FUNCTION_BLOCK ButtonColorChanger (* Composite FB wrapping other FBs *)
  (* Standard: 61499-2 *)
  (* Version 1.0, 2022-08-01, franz *)
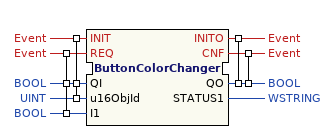
  EVENT_INPUT
    INIT WITH QI, u16ObjId; (* Initialization Request *)
    REQ WITH QI, I1; (* Normal Execution Request *)
  END_EVENT
  EVENT_OUTPUT
    INITO WITH QO; (* Initialization Confirm *)
    CNF WITH QO; (* Execution Confirmation *)
  END_EVENT
  VAR_INPUT
    QI : BOOL; (* Input event qualifier *)
    u16ObjId : UINT; (* Object ID *)
    I1 : BOOL;
  END_VAR
  VAR_OUTPUT
    QO : BOOL; (* Output event qualifier *)
    STATUS1 : WSTRING;
  END_VAR
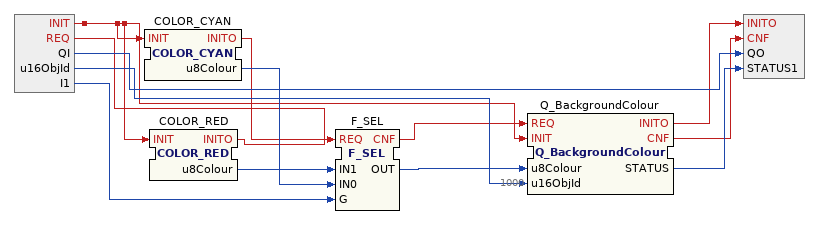
  FBS
    Q_BackgroundColour : Q_BackgroundColour(u16ObjId := 1000);
    F_SEL : F_SEL;
    COLOR_RED : COLOR_RED;
    COLOR_CYAN : COLOR_CYAN;
  END_FBS
  EVENT_CONNECTIONS
    F_SEL.CNF TO Q_BackgroundColour.REQ;
    COLOR_CYAN.INITO TO F_SEL.REQ;
    COLOR_RED.INITO TO F_SEL.REQ;
    Q_BackgroundColour.INITO TO INITO;
    INIT TO COLOR_CYAN.INIT;
    INIT TO COLOR_RED.INIT;
    Q_BackgroundColour.CNF TO CNF;
    REQ TO F_SEL.REQ;
    INIT TO Q_BackgroundColour.INIT;
  END_CONNECTIONS
  DATA_CONNECTIONS
    COLOR_RED.u8Colour TO F_SEL.IN1;
    COLOR_CYAN.u8Colour TO F_SEL.IN0;
    F_SEL.OUT TO Q_BackgroundColour.u8Colour;
    u16ObjId TO Q_BackgroundColour.u16ObjId;
    Q_BackgroundColour.STATUS TO STATUS1;
    QI TO QO;
    I1 TO F_SEL.G;
  END_CONNECTIONS
END_FUNCTION_BLOCK
